// SIMATIC S7-200 project (STEP 7-Micro/WIN), CPU 224 AM REL 21.02

SYMBOL_TABLE USER1
T2SK1_TG         C1
T2SK2_TG         C2
T2SK3_TG         C3
T2SK4_TG         C4
T2SK5_TG         C5
T2SK6_TG         C6
T2SK7_TG         C7
T2SK8_TG         C8
T2SK9_TG         C9
T3SK1_TG         C10
T3SK2_TG         C11
T3SK3_TG         C12
T3SK4_TG         C13
T3SK5_TG         C14
T3SK6_TG         C15
T3SK7_TG         C16
T3SK8_TG         C17
T3SK9_TG         C18
T4SK1_TG         C19
T4SK2_TG         C20
T4SK3_TG         C21
T4SK4_TG         C22
T4SK5_TG         C23
T4SK6_TG         C24
T4SK7_TG         C25
T4SK8_TG         C26
T4SK9_TG         C27
T5SK1_TG         C28
T5SK2_TG         C29
T5SK3_TG         C30
T5SK4_TG         C31
T5SK5_TG         C32
T5SK6_TG         C33
T5SK7_TG         C34
T5SK8_TG         C35
T5SK9_TG         C36
T6SK1_TG         C37
T6SK2_TG         C38
T6SK3_TG         C39
T6SK4_TG         C40
T6SK5_TG         C41
T6SK6_TG         C42
T6SK7_TG         C43
T6SK8_TG         C44
T6SK9_TG         C45
T7SK1_TG         C46
T7SK2_TG         C47
T7SK3_TG         C48
T7SK4_TG         C49
T7SK5_TG         C50
T7SK6_TG         C51
T7SK7_TG         C52
T7SK8_TG         C53
T7SK9_TG         C54
CNSK1_TG         C55
CNSK2_TG         C56
CNSK3_TG         C57
CNSK4_TG         C58
CNSK5_TG         C59
CNSK6_TG         C60
CNSK7_TG         C61
CNSK8_TG         C62
CNSK9_TG         C63
GIO              MW0
NGAY             MW2
PHUT             MW4
THANG            MW6
THU              MW8
GIAY             MW10
AT1              Q0.0
AT2              Q0.1
AT3              Q0.2
AT4              Q0.3
AT5              Q0.4
AT6              Q0.5
AT7              Q0.6
AT8              Q0.7
TEST_1           V10.0
TEST_2           V10.1
TEST_3           V10.2
TEST_4           V10.3
TEST_5           V10.4
TEST_6           V10.5
TEST_7           V10.6
TEST_8           V10.7
T2RS             V11.2
GOI_AT           V11.3
T3RS             V11.4
T4RS             V11.5
T5RS             V11.6
T6RS             V11.7
T7RS             V12.0
CNRS             V12.1
T2SK1H           VW100
T2SK1M           VW102
T2SK1LC          VW104
T2SK1_TGD        VW106
T2SK2H           VW108
T2SK2M           VW110
T2SK2LC          VW112
T2SK2_TGD        VW114
T2SK3H           VW116
T2SK3M           VW118
T2SK3LC          VW120
T2SK3_TGD        VW122
T2SK4H           VW124
T2SK4M           VW126
T2SK4LC          VW128
T2SK4_TGD        VW130
T2SK5H           VW132
T2SK5M           VW134
T2SK5LC          VW136
T2SK5_TGD        VW138
T2SK6H           VW140
T2SK6M           VW142
T2SK6LC          VW144
T2SK6_TGD        VW146
T2SK7H           VW148
T2SK7M           VW150
T2SK7LC          VW152
T2SK7_TGD        VW154
T2SK8H           VW156
T2SK8M           VW158
T2SK8LC          VW160
T2SK8_TGD        VW162
T2SK9H           VW164
T2SK9M           VW166
T2SK9LC          VW168
T2SK9_TGD        VW170
T3SK1H           VW172
T3SK1M           VW174
T3SK1LC          VW176
T3SK1_TGD        VW178
T3SK2H           VW180
T3SK2M           VW182
T3SK2LC          VW184
T3SK2_TGD        VW186
T3SK3H           VW188
T3SK3M           VW190
T3SK3LC          VW192
T3SK3_TGD        VW194
T3SK4H           VW196
T3SK4M           VW198
T3SK4LC          VW200
T3SK4_TGD        VW202
T3SK5H           VW204
T3SK5M           VW206
T3SK5LC          VW208
T3SK5_TGD        VW210
T3SK6H           VW212
T3SK6M           VW214
T3SK6LC          VW216
T3SK6_TGD        VW218
T3SK7H           VW220
T3SK7M           VW222
T3SK7LC          VW224
T3SK7_TGD        VW226
T3SK8H           VW228
T3SK8M           VW230
T3SK8LC          VW232
T3SK8_TGD        VW234
T3SK9H           VW236
T3SK9M           VW238
T3SK9LC          VW240
T3SK9_TGD        VW242
T4SK1H           VW244
T4SK1M           VW246
T4SK1LC          VW248
T4SK1_TGD        VW250
T4SK2H           VW252
T4SK2M           VW254
T4SK2LC          VW256
T4SK2_TGD        VW258
T4SK3H           VW260
T4SK3M           VW262
T4SK3LC          VW264
T4SK3_TGD        VW266
T4SK4H           VW268
T4SK4M           VW270
T4SK4LC          VW272
T4SK4_TGD        VW274
T4SK5H           VW276
T4SK5M           VW278
T4SK5LC          VW280
T4SK5_TGD        VW282
T4SK6H           VW284
T4SK6M           VW286
T4SK6LC          VW288
T4SK6_TGD        VW290
T4SK7H           VW292
T4SK7M           VW294
T4SK7LC          VW296
T4SK7_TGD        VW298
T4SK8H           VW300
T4SK8M           VW302
T4SK8LC          VW304
T4SK8_TGD        VW306
T4SK9H           VW308
T4SK9M           VW310
T4SK9LC          VW312
T4SK9_TGD        VW314
T5SK1H           VW316
T5SK1M           VW318
T5SK1LC          VW320
T5SK1_TGD        VW322
T5SK2H           VW324
T5SK2M           VW326
T5SK2LC          VW328
T5SK2_TGD        VW330
T5SK3H           VW332
T5SK3M           VW334
T5SK3LC          VW336
T5SK3_TGD        VW338
T5SK4H           VW340
T5SK4M           VW342
T5SK4LC          VW346
T5SK4_TGD        VW348
T5SK5H           VW350
T5SK5M           VW352
T5SK5LC          VW354
T5SK5_TGD        VW356
T5SK6H           VW358
T5SK6M           VW360
T5SK6LC          VW362
T5SK6_TGD        VW364
T5SK7H           VW368
T5SK7M           VW370
T5SK7LC          VW372
T5SK7_TGD        VW374
T5SK8H           VW376
T5SK8M           VW378
T5SK8LC          VW380
T5SK8_TGD        VW382
T5SK9H           VW384
T5SK9M           VW386
T5SK9LC          VW388
T5SK9_TGD        VW390
T6SK1H           VW392
T6SK1M           VW394
T6SK1LC          VW396
T6SK1_TGD        VW398
T6SK2H           VW400
T6SK2M           VW402
T6SK2LC          VW404
T6SK2_TGD        VW406
T6SK3H           VW408
T6SK3M           VW410
T6SK3LC          VW412
T6SK3_TGD        VW414
T6SK4H           VW416
T6SK4M           VW418
T6SK4LC          VW420
T6SK4_TGD        VW422
T6SK5H           VW424
T6SK5M           VW426
T6SK5LC          VW428
T6SK5_TGD        VW430
T6SK6H           VW432
T6SK6M           VW434
T6SK6LC          VW436
T6SK6_TGD        VW438
T6SK7H           VW440
T6SK7M           VW442
T6SK7LC          VW444
T6SK7_TGD        VW446
T6SK8H           VW448
T6SK8M           VW450
T6SK8LC          VW452
T6SK8_TGD        VW454
T6SK9H           VW456
T6SK9M           VW458
T6SK9LC          VW460
T6SK9_TGD        VW462
T7SK1H           VW468
T7SK1M           VW470
T7SK1LC          VW472
T7SK1_TGD        VW474
T7SK2H           VW476
T7SK2M           VW478
T7SK2LC          VW480
T7SK2_TGD        VW482
T7SK3H           VW484
T7SK3M           VW486
T7SK3LC          VW488
T7SK3_TGD        VW490
T7SK4H           VW492
T7SK4M           VW494
T7SK4LC          VW496
T7SK4_TGD        VW498
T7SK5H           VW500
T7SK5M           VW502
T7SK5LC          VW504
T7SK5_TGD        VW506
T7SK6H           VW508
T7SK6M           VW510
T7SK6LC          VW512
T7SK6_TGD        VW514
T7SK7H           VW516
T7SK7M           VW518
T7SK7LC          VW520
T7SK7_TGD        VW522
T7SK8H           VW524
T7SK8M           VW526
T7SK8LC          VW528
T7SK8_TGD        VW530
T7SK9H           VW532
T7SK9M           VW534
T7SK9LC          VW536
T7SK9_TGD        VW538
CNSK1H           VW540
CNSK1M           VW542
CNSK1LC          VW546
CNSK1_TGD        VW548
CNSK2H           VW550
CNSK2M           VW552
CNSK2LC          VW554
CNSK2_TGD        VW556
CNSK3H           VW558
CNSK3M           VW560
CNSK3LC          VW562
CNSK3_TGD        VW564
CNSK4H           VW566
CNSK4M           VW568
CNSK4LC          VW570
CNSK4_TGD        VW572
CNSK5H           VW574
CNSK5M           VW576
CNSK5LC          VW578
CNSK5_TGD        VW580
CNSK6H           VW582
CNSK6M           VW584
CNSK6LC          VW586
CNSK6_TGD        VW588
CNSK7H           VW590
CNSK7M           VW592
CNSK7LC          VW594
CNSK7_TGD        VW596
CNSK8H           VW598
CNSK8M           VW600
CNSK8LC          VW602
CNSK8_TGD        VW604
CNSK9H           VW606
CNSK9M           VW608
CNSK9LC          VW610
CNSK9_TGD        VW612
END_SYMBOL_TABLE

ORGANIZATION_BLOCK MAIN:OB1
TITLE=PROGRAM COMMENTS
BEGIN
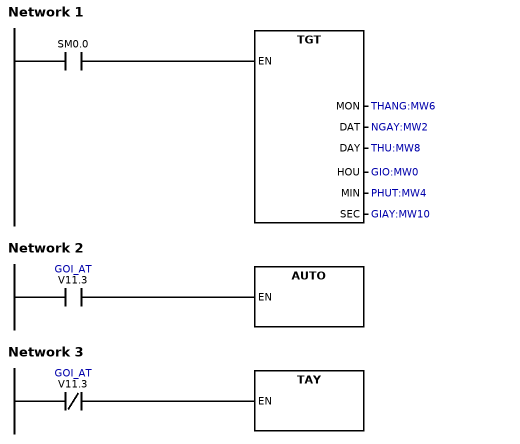
Network 1
LD     SM0.0
CALL   TGT:SBR0, THANG:MW6, NGAY:MW2, THU:MW8, GIO:MW0, PHUT:MW4, GIAY:MW10
Network 2
LD     GOI_AT:V11.3
CALL   AUTO:SBR2
Network 3
LDN    GOI_AT:V11.3
CALL   TAY:SBR1
END_ORGANIZATION_BLOCK

SUBROUTINE_BLOCK TGT:SBR0
TITLE=SUBROUTINE COMMENTS
VAR_OUTPUT
MON:INT;	// LW0 
DAT:INT;	// LW2 
DAY:INT;	// LW4 
HOU:INT;	// LW6 
MIN:INT;	// LW8 
SEC:INT;	// LW10 
END_VAR
BEGIN
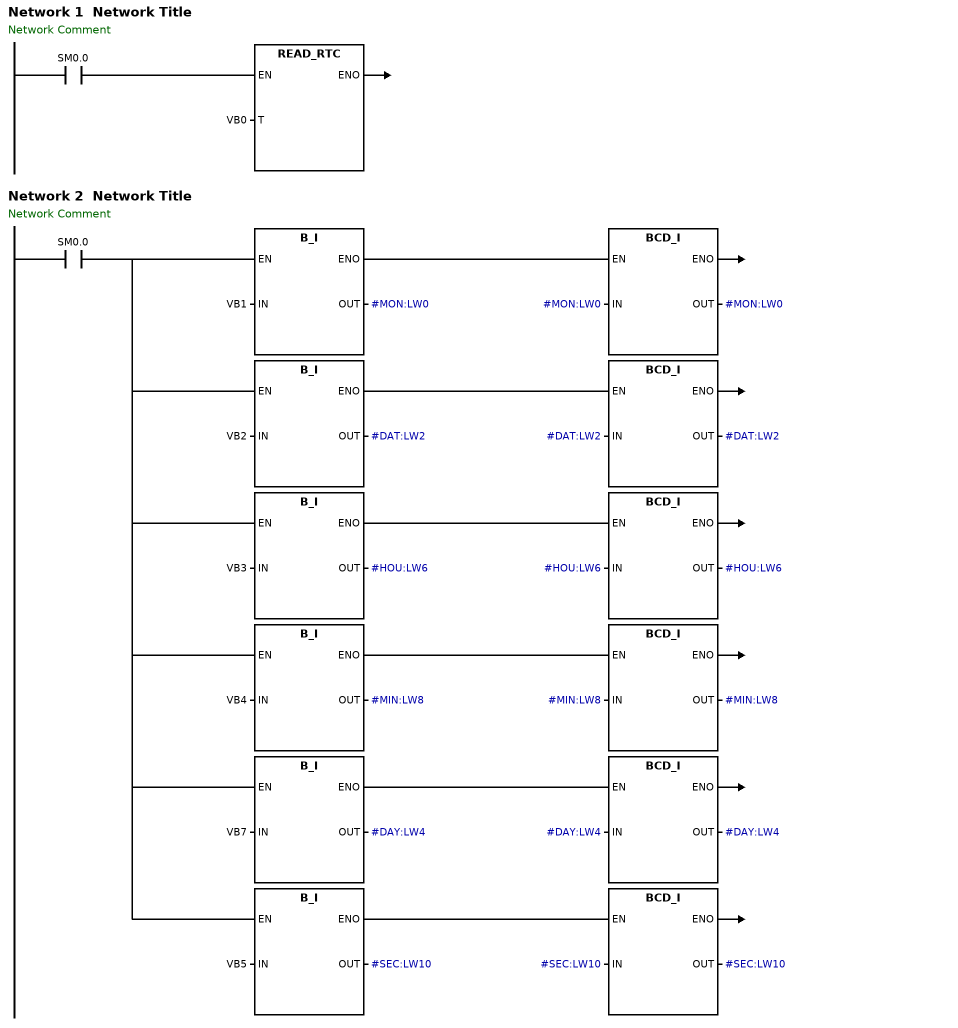
Network 1 // Network Title
// Network Comment
LD     SM0.0
TODR   VB0
Network 2 // Network Title
// Network Comment
LD     SM0.0
LPS
BTI    VB1, #MON:LW0
AENO
BCDI   #MON:LW0
LRD
BTI    VB2, #DAT:LW2
AENO
BCDI   #DAT:LW2
LRD
BTI    VB3, #HOU:LW6
AENO
BCDI   #HOU:LW6
LRD
BTI    VB4, #MIN:LW8
AENO
BCDI   #MIN:LW8
LRD
BTI    VB7, #DAY:LW4
AENO
BCDI   #DAY:LW4
LPP
BTI    VB5, #SEC:LW10
AENO
BCDI   #SEC:LW10
END_SUBROUTINE_BLOCK

SUBROUTINE_BLOCK TAY:SBR1
TITLE=SUBROUTINE COMMENTS
BEGIN
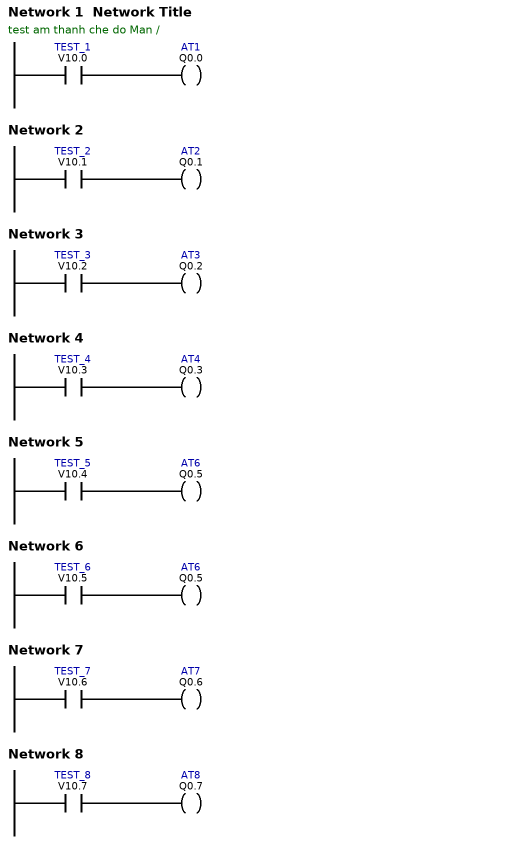
Network 1 // Network Title
// test am thanh che do Man
// 
LD     TEST_1:V10.0
=      AT1:Q0.0
Network 2
LD     TEST_2:V10.1
=      AT2:Q0.1
Network 3
LD     TEST_3:V10.2
=      AT3:Q0.2
Network 4
LD     TEST_4:V10.3
=      AT4:Q0.3
Network 5
LD     TEST_5:V10.4
=      AT6:Q0.5
Network 6
LD     TEST_6:V10.5
=      AT6:Q0.5
Network 7
LD     TEST_7:V10.6
=      AT7:Q0.6
Network 8
LD     TEST_8:V10.7
=      AT8:Q0.7
END_SUBROUTINE_BLOCK

SUBROUTINE_BLOCK AUTO:SBR2
TITLE=SUBROUTINE COMMENTS
BEGIN
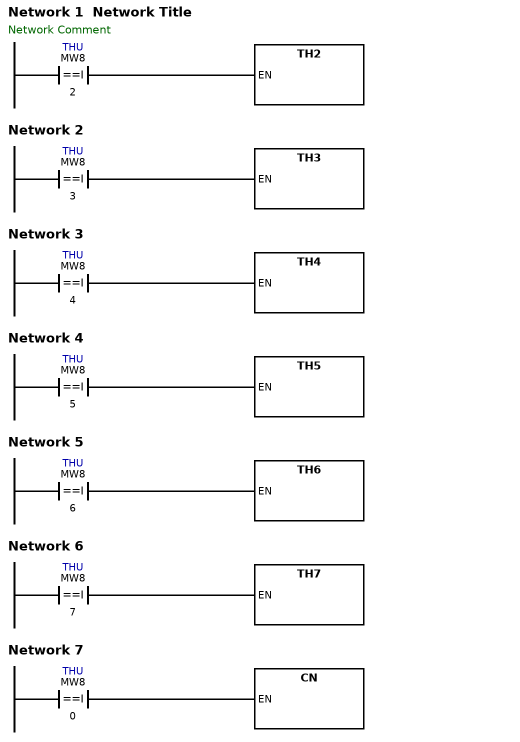
Network 1 // Network Title
// Network Comment
LDW=   THU:MW8, 2
CALL   TH2:SBR3
Network 2
LDW=   THU:MW8, 3
CALL   TH3:SBR4
Network 3
LDW=   THU:MW8, 4
CALL   TH4:SBR5
Network 4
LDW=   THU:MW8, 5
CALL   TH5:SBR6
Network 5
LDW=   THU:MW8, 6
CALL   TH6:SBR7
Network 6
LDW=   THU:MW8, 7
CALL   TH7:SBR8
Network 7
LDW=   THU:MW8, 0
CALL   CN:SBR9
END_SUBROUTINE_BLOCK

SUBROUTINE_BLOCK TH2:SBR3
TITLE=SUBROUTINE COMMENTS
VAR
TAM1:BOOL;	// L0.0 
TAM2:BOOL;	// L0.1 
TAM3:BOOL;	// L0.2 
TAM4:BOOL;	// L0.3 
TAM5:BOOL;	// L0.4 
TAM6:BOOL;	// L0.5 
TAM7:BOOL;	// L0.6 
TAM8:BOOL;	// L0.7 
TAM9:BOOL;	// L1.0 
END_VAR
BEGIN
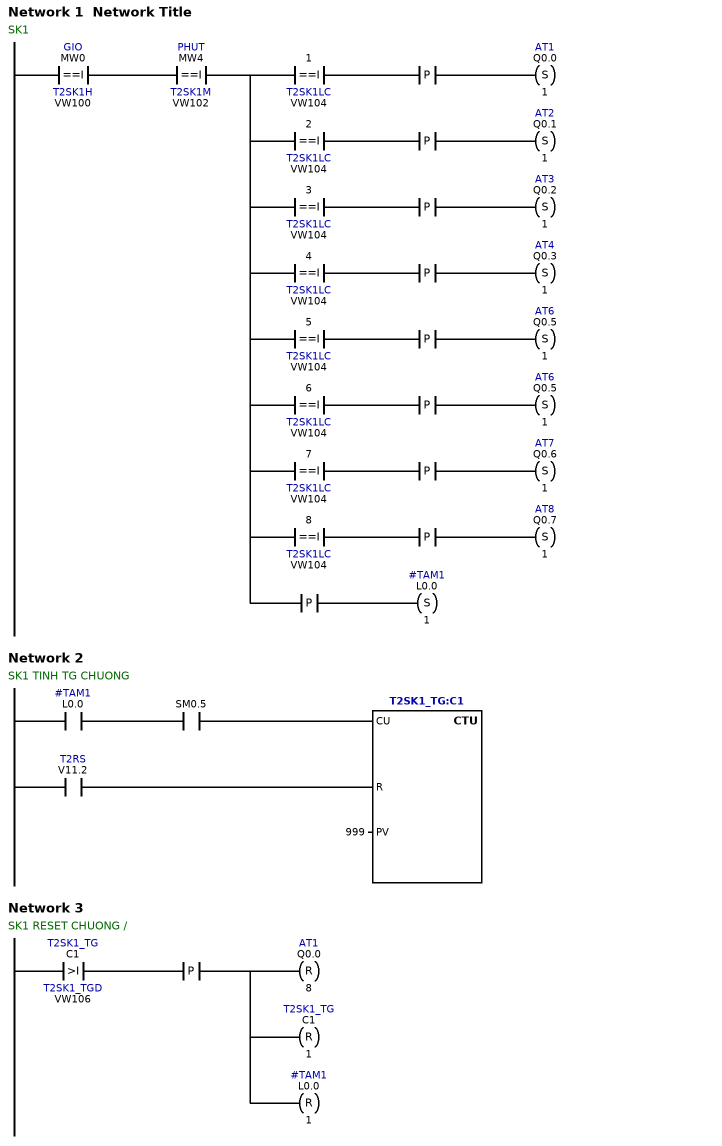
Network 1 // Network Title
// SK1	
LDW=   GIO:MW0, T2SK1H:VW100
AW=    PHUT:MW4, T2SK1M:VW102
LPS
AW=    1, T2SK1LC:VW104
EU
S      AT1:Q0.0, 1
LRD
AW=    2, T2SK1LC:VW104
EU
S      AT2:Q0.1, 1
LRD
AW=    3, T2SK1LC:VW104
EU
S      AT3:Q0.2, 1
LRD
AW=    4, T2SK1LC:VW104
EU
S      AT4:Q0.3, 1
LRD
AW=    5, T2SK1LC:VW104
EU
S      AT6:Q0.5, 1
LRD
AW=    6, T2SK1LC:VW104
EU
S      AT6:Q0.5, 1
LRD
AW=    7, T2SK1LC:VW104
EU
S      AT7:Q0.6, 1
LRD
AW=    8, T2SK1LC:VW104
EU
S      AT8:Q0.7, 1
LPP
EU
S      #TAM1:L0.0, 1
Network 2
// SK1 TINH TG CHUONG
LD     #TAM1:L0.0
A      SM0.5
LD     T2RS:V11.2
CTU    T2SK1_TG:C1, 999
Network 3
// SK1 RESET CHUONG
// 
LDW>   T2SK1_TG:C1, T2SK1_TGD:VW106
EU
R      AT1:Q0.0, 8
R      T2SK1_TG:C1, 1
R      #TAM1:L0.0, 1
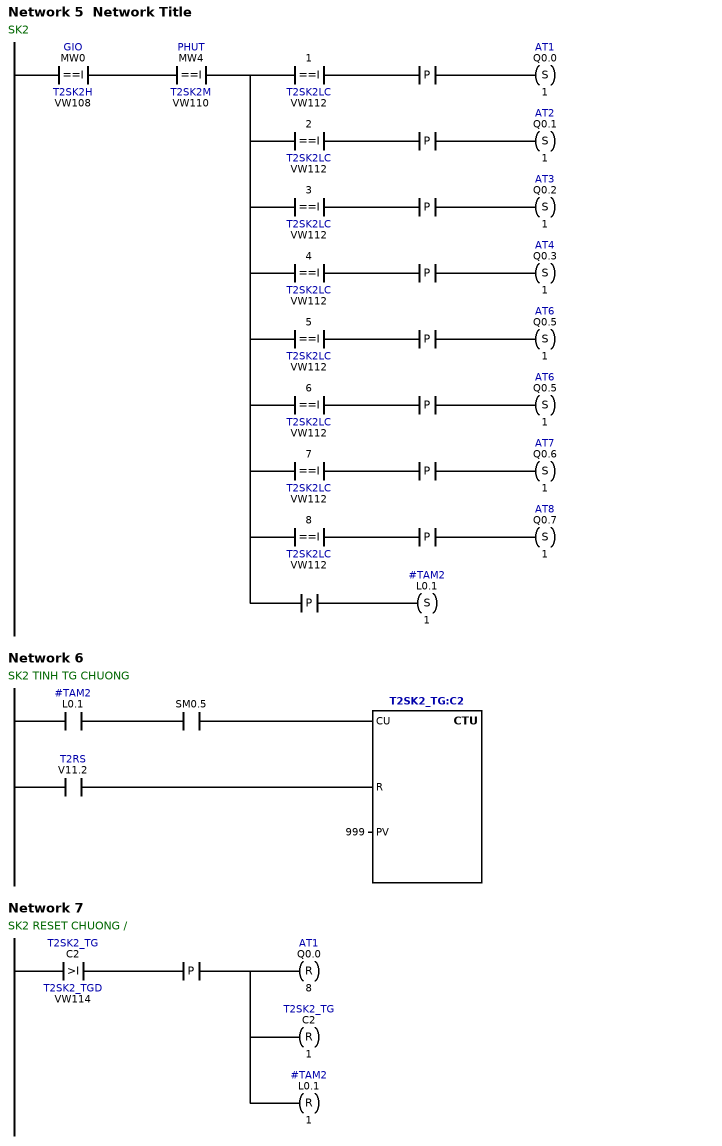
Network 5 // Network Title
// SK2
LDW=   GIO:MW0, T2SK2H:VW108
AW=    PHUT:MW4, T2SK2M:VW110
LPS
AW=    1, T2SK2LC:VW112
EU
S      AT1:Q0.0, 1
LRD
AW=    2, T2SK2LC:VW112
EU
S      AT2:Q0.1, 1
LRD
AW=    3, T2SK2LC:VW112
EU
S      AT3:Q0.2, 1
LRD
AW=    4, T2SK2LC:VW112
EU
S      AT4:Q0.3, 1
LRD
AW=    5, T2SK2LC:VW112
EU
S      AT6:Q0.5, 1
LRD
AW=    6, T2SK2LC:VW112
EU
S      AT6:Q0.5, 1
LRD
AW=    7, T2SK2LC:VW112
EU
S      AT7:Q0.6, 1
LRD
AW=    8, T2SK2LC:VW112
EU
S      AT8:Q0.7, 1
LPP
EU
S      #TAM2:L0.1, 1
Network 6
// SK2 TINH TG CHUONG
LD     #TAM2:L0.1
A      SM0.5
LD     T2RS:V11.2
CTU    T2SK2_TG:C2, 999
Network 7
// SK2 RESET CHUONG
// 
LDW>   T2SK2_TG:C2, T2SK2_TGD:VW114
EU
R      AT1:Q0.0, 8
R      T2SK2_TG:C2, 1
R      #TAM2:L0.1, 1
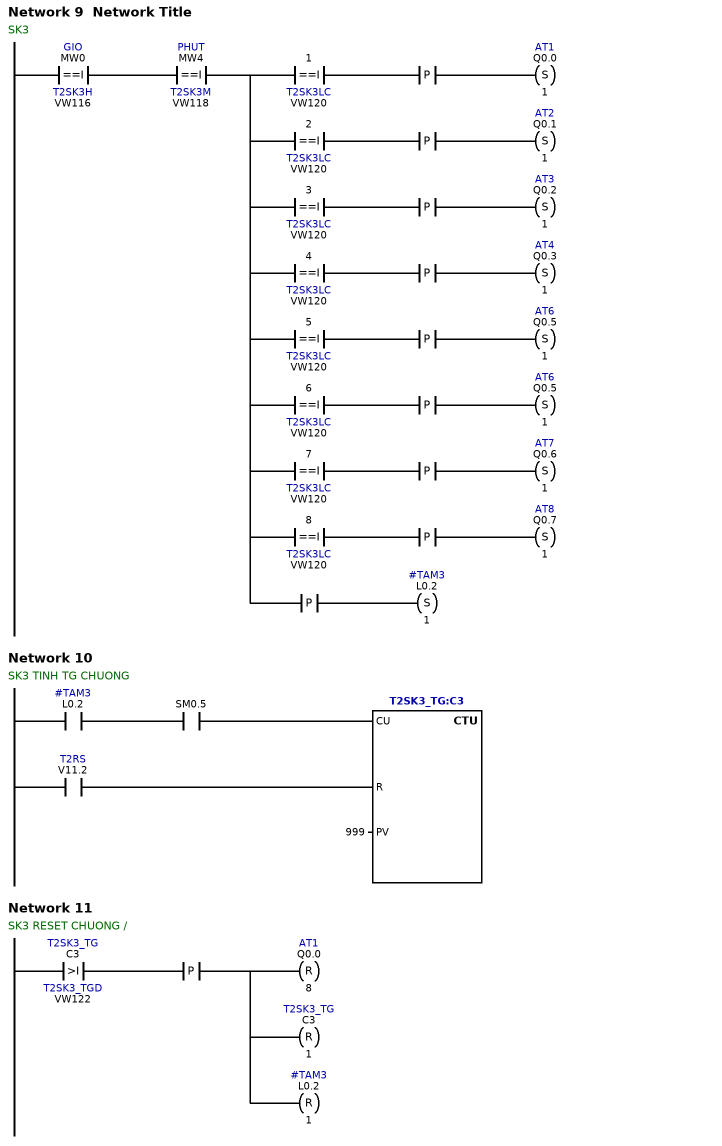
Network 9 // Network Title
// SK3	
LDW=   GIO:MW0, T2SK3H:VW116
AW=    PHUT:MW4, T2SK3M:VW118
LPS
AW=    1, T2SK3LC:VW120
EU
S      AT1:Q0.0, 1
LRD
AW=    2, T2SK3LC:VW120
EU
S      AT2:Q0.1, 1
LRD
AW=    3, T2SK3LC:VW120
EU
S      AT3:Q0.2, 1
LRD
AW=    4, T2SK3LC:VW120
EU
S      AT4:Q0.3, 1
LRD
AW=    5, T2SK3LC:VW120
EU
S      AT6:Q0.5, 1
LRD
AW=    6, T2SK3LC:VW120
EU
S      AT6:Q0.5, 1
LRD
AW=    7, T2SK3LC:VW120
EU
S      AT7:Q0.6, 1
LRD
AW=    8, T2SK3LC:VW120
EU
S      AT8:Q0.7, 1
LPP
EU
S      #TAM3:L0.2, 1
Network 10
// SK3 TINH TG CHUONG
LD     #TAM3:L0.2
A      SM0.5
LD     T2RS:V11.2
CTU    T2SK3_TG:C3, 999
Network 11
// SK3 RESET CHUONG
// 
LDW>   T2SK3_TG:C3, T2SK3_TGD:VW122
EU
R      AT1:Q0.0, 8
R      T2SK3_TG:C3, 1
R      #TAM3:L0.2, 1
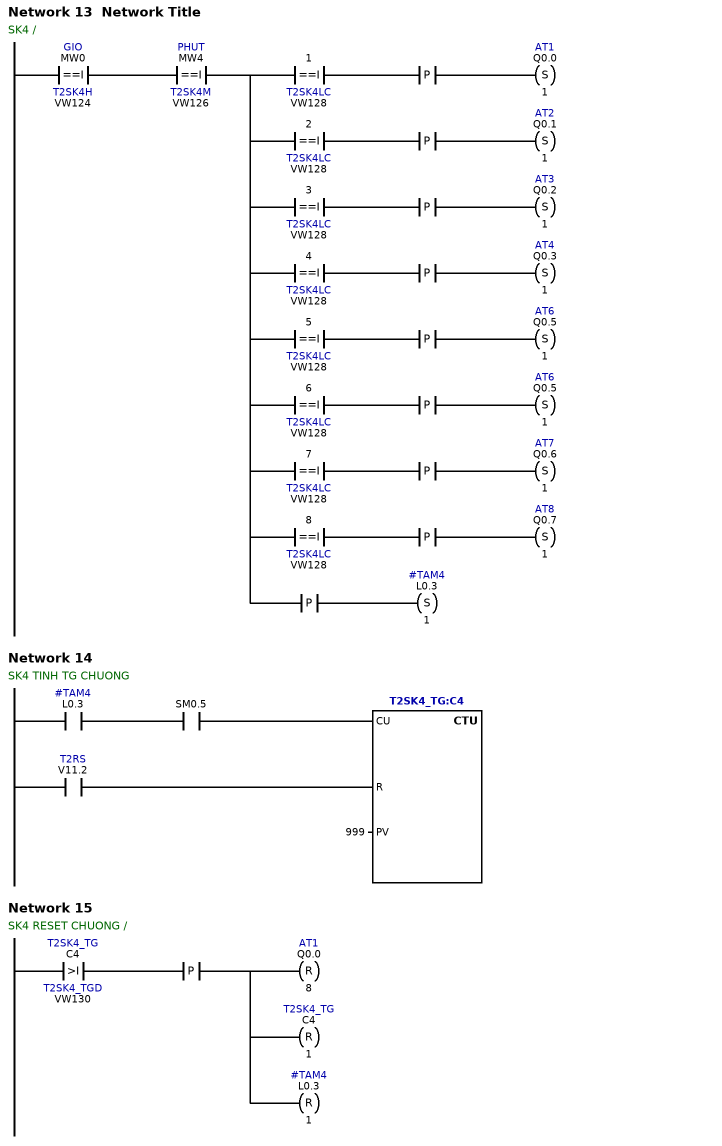
Network 13 // Network Title
// SK4
// 	
LDW=   GIO:MW0, T2SK4H:VW124
AW=    PHUT:MW4, T2SK4M:VW126
LPS
AW=    1, T2SK4LC:VW128
EU
S      AT1:Q0.0, 1
LRD
AW=    2, T2SK4LC:VW128
EU
S      AT2:Q0.1, 1
LRD
AW=    3, T2SK4LC:VW128
EU
S      AT3:Q0.2, 1
LRD
AW=    4, T2SK4LC:VW128
EU
S      AT4:Q0.3, 1
LRD
AW=    5, T2SK4LC:VW128
EU
S      AT6:Q0.5, 1
LRD
AW=    6, T2SK4LC:VW128
EU
S      AT6:Q0.5, 1
LRD
AW=    7, T2SK4LC:VW128
EU
S      AT7:Q0.6, 1
LRD
AW=    8, T2SK4LC:VW128
EU
S      AT8:Q0.7, 1
LPP
EU
S      #TAM4:L0.3, 1
Network 14
// SK4 TINH TG CHUONG
LD     #TAM4:L0.3
A      SM0.5
LD     T2RS:V11.2
CTU    T2SK4_TG:C4, 999
Network 15
// SK4 RESET CHUONG
// 
LDW>   T2SK4_TG:C4, T2SK4_TGD:VW130
EU
R      AT1:Q0.0, 8
R      T2SK4_TG:C4, 1
R      #TAM4:L0.3, 1
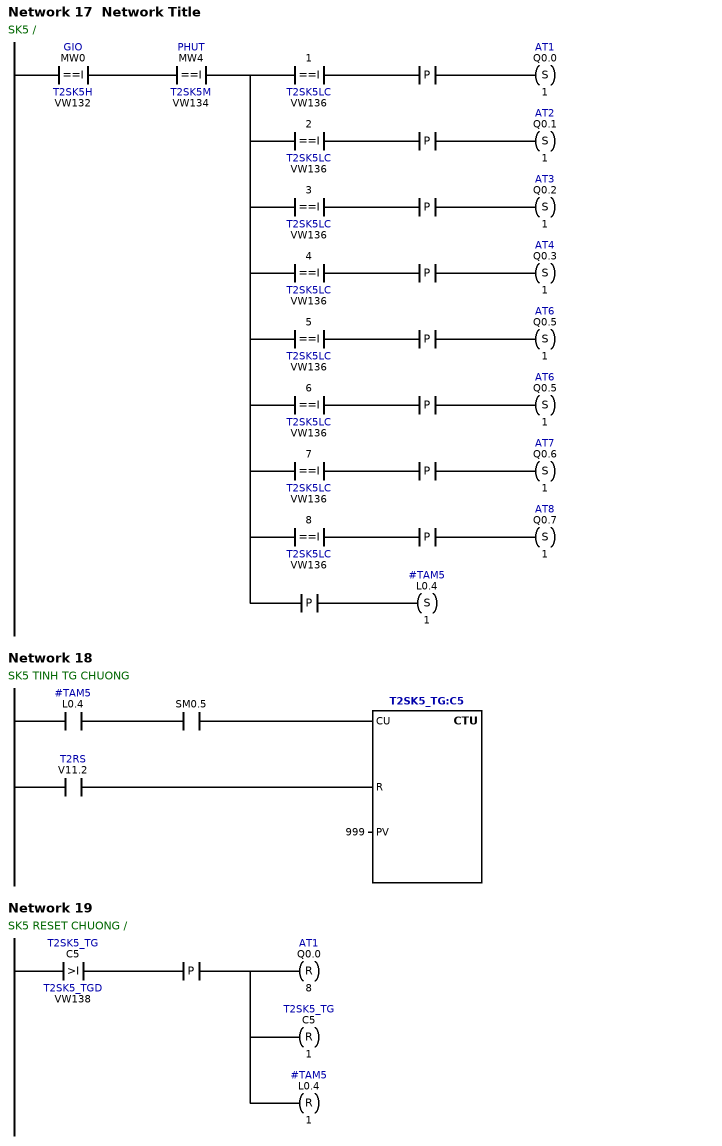
Network 17 // Network Title
// SK5
// 	
LDW=   GIO:MW0, T2SK5H:VW132
AW=    PHUT:MW4, T2SK5M:VW134
LPS
AW=    1, T2SK5LC:VW136
EU
S      AT1:Q0.0, 1
LRD
AW=    2, T2SK5LC:VW136
EU
S      AT2:Q0.1, 1
LRD
AW=    3, T2SK5LC:VW136
EU
S      AT3:Q0.2, 1
LRD
AW=    4, T2SK5LC:VW136
EU
S      AT4:Q0.3, 1
LRD
AW=    5, T2SK5LC:VW136
EU
S      AT6:Q0.5, 1
LRD
AW=    6, T2SK5LC:VW136
EU
S      AT6:Q0.5, 1
LRD
AW=    7, T2SK5LC:VW136
EU
S      AT7:Q0.6, 1
LRD
AW=    8, T2SK5LC:VW136
EU
S      AT8:Q0.7, 1
LPP
EU
S      #TAM5:L0.4, 1
Network 18
// SK5 TINH TG CHUONG
LD     #TAM5:L0.4
A      SM0.5
LD     T2RS:V11.2
CTU    T2SK5_TG:C5, 999
Network 19
// SK5 RESET CHUONG
// 
LDW>   T2SK5_TG:C5, T2SK5_TGD:VW138
EU
R      AT1:Q0.0, 8
R      T2SK5_TG:C5, 1
R      #TAM5:L0.4, 1
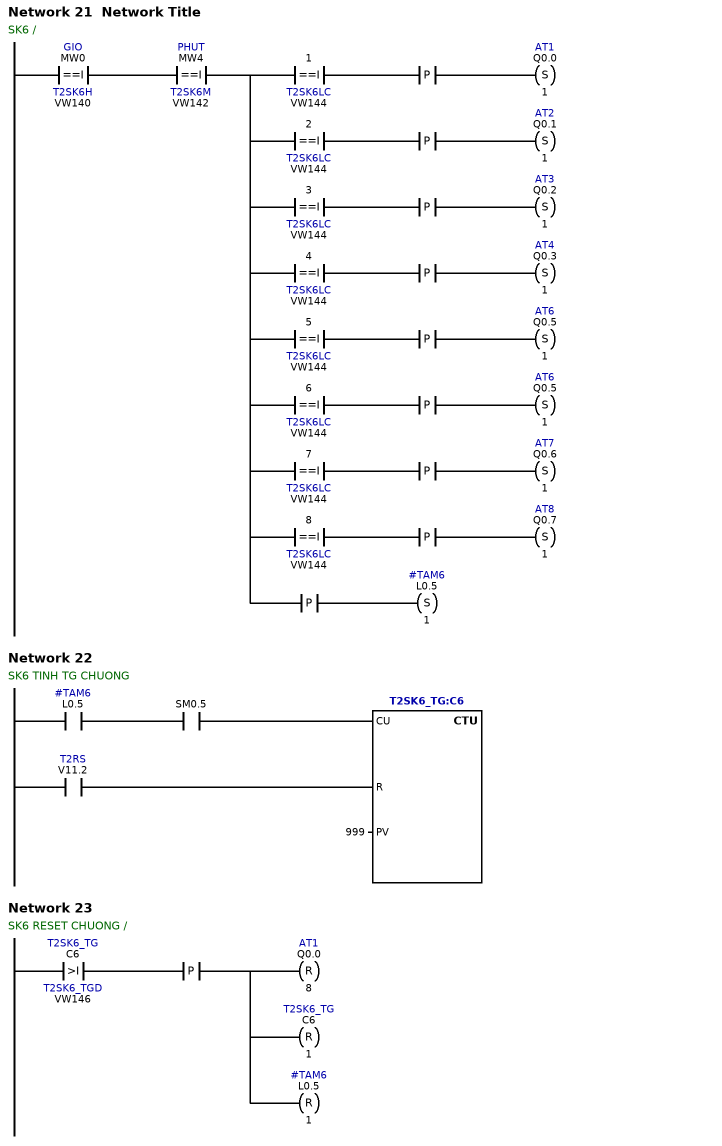
Network 21 // Network Title
// SK6
// 	
LDW=   GIO:MW0, T2SK6H:VW140
AW=    PHUT:MW4, T2SK6M:VW142
LPS
AW=    1, T2SK6LC:VW144
EU
S      AT1:Q0.0, 1
LRD
AW=    2, T2SK6LC:VW144
EU
S      AT2:Q0.1, 1
LRD
AW=    3, T2SK6LC:VW144
EU
S      AT3:Q0.2, 1
LRD
AW=    4, T2SK6LC:VW144
EU
S      AT4:Q0.3, 1
LRD
AW=    5, T2SK6LC:VW144
EU
S      AT6:Q0.5, 1
LRD
AW=    6, T2SK6LC:VW144
EU
S      AT6:Q0.5, 1
LRD
AW=    7, T2SK6LC:VW144
EU
S      AT7:Q0.6, 1
LRD
AW=    8, T2SK6LC:VW144
EU
S      AT8:Q0.7, 1
LPP
EU
S      #TAM6:L0.5, 1
Network 22
// SK6 TINH TG CHUONG
LD     #TAM6:L0.5
A      SM0.5
LD     T2RS:V11.2
CTU    T2SK6_TG:C6, 999
Network 23
// SK6 RESET CHUONG
// 
LDW>   T2SK6_TG:C6, T2SK6_TGD:VW146
EU
R      AT1:Q0.0, 8
R      T2SK6_TG:C6, 1
R      #TAM6:L0.5, 1
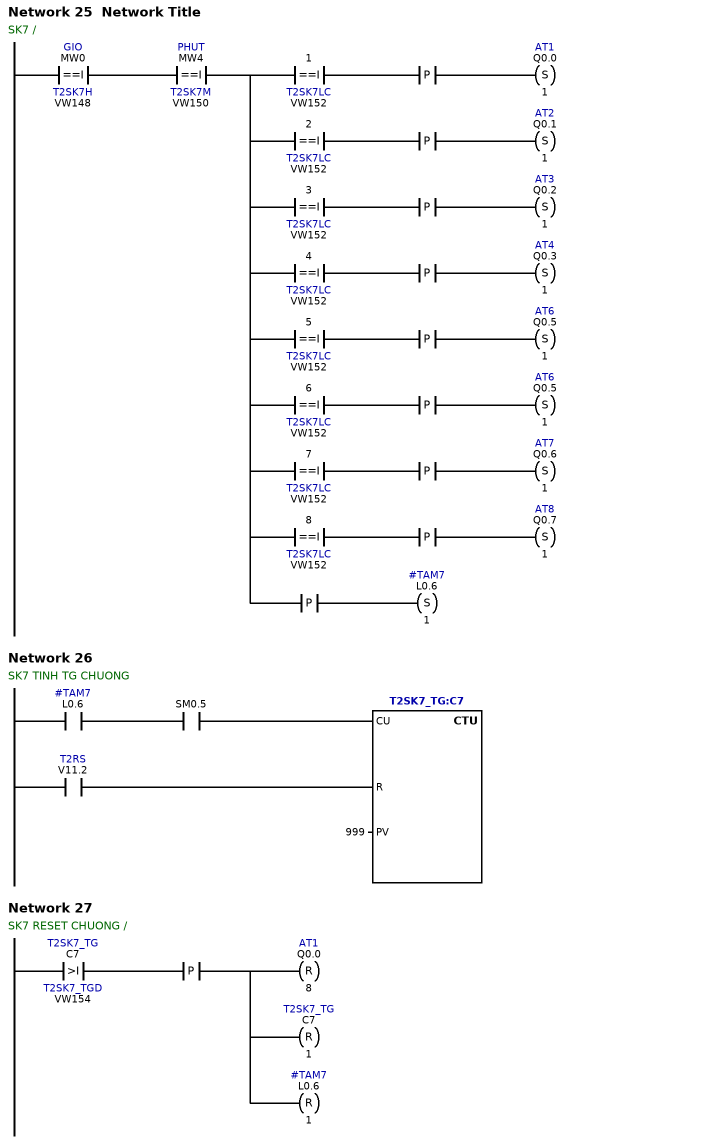
Network 25 // Network Title
// SK7
// 	
LDW=   GIO:MW0, T2SK7H:VW148
AW=    PHUT:MW4, T2SK7M:VW150
LPS
AW=    1, T2SK7LC:VW152
EU
S      AT1:Q0.0, 1
LRD
AW=    2, T2SK7LC:VW152
EU
S      AT2:Q0.1, 1
LRD
AW=    3, T2SK7LC:VW152
EU
S      AT3:Q0.2, 1
LRD
AW=    4, T2SK7LC:VW152
EU
S      AT4:Q0.3, 1
LRD
AW=    5, T2SK7LC:VW152
EU
S      AT6:Q0.5, 1
LRD
AW=    6, T2SK7LC:VW152
EU
S      AT6:Q0.5, 1
LRD
AW=    7, T2SK7LC:VW152
EU
S      AT7:Q0.6, 1
LRD
AW=    8, T2SK7LC:VW152
EU
S      AT8:Q0.7, 1
LPP
EU
S      #TAM7:L0.6, 1
Network 26
// SK7 TINH TG CHUONG
LD     #TAM7:L0.6
A      SM0.5
LD     T2RS:V11.2
CTU    T2SK7_TG:C7, 999
Network 27
// SK7 RESET CHUONG
// 
LDW>   T2SK7_TG:C7, T2SK7_TGD:VW154
EU
R      AT1:Q0.0, 8
R      T2SK7_TG:C7, 1
R      #TAM7:L0.6, 1
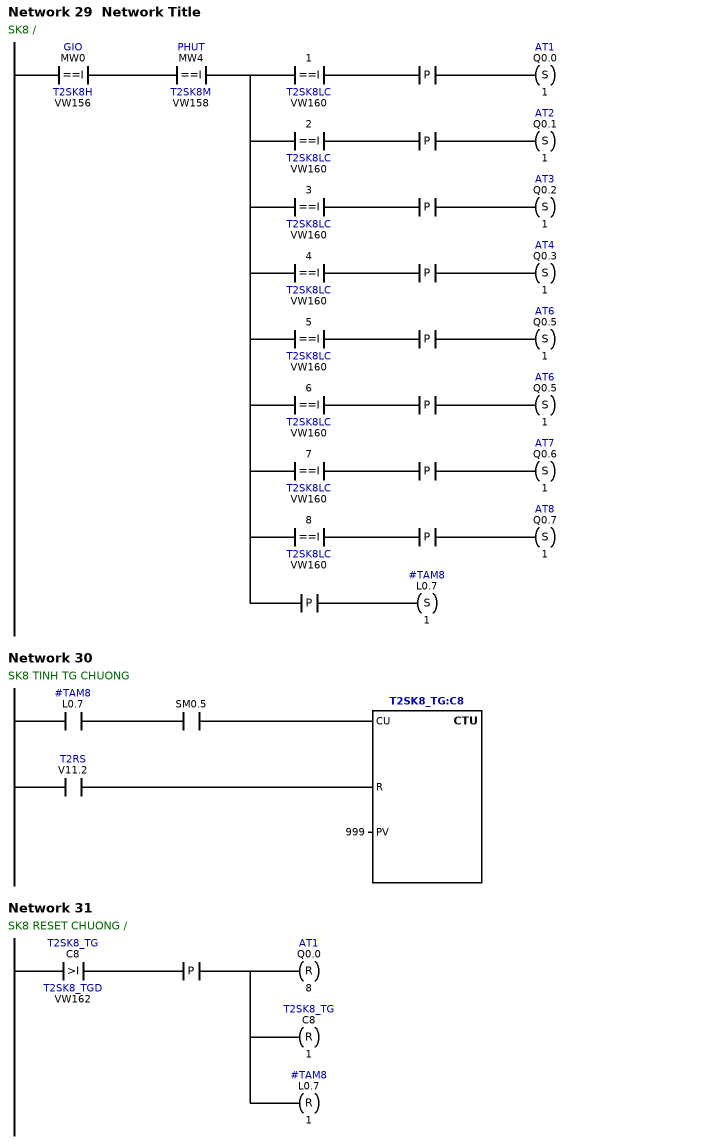
Network 29 // Network Title
// SK8
// 	
LDW=   GIO:MW0, T2SK8H:VW156
AW=    PHUT:MW4, T2SK8M:VW158
LPS
AW=    1, T2SK8LC:VW160
EU
S      AT1:Q0.0, 1
LRD
AW=    2, T2SK8LC:VW160
EU
S      AT2:Q0.1, 1
LRD
AW=    3, T2SK8LC:VW160
EU
S      AT3:Q0.2, 1
LRD
AW=    4, T2SK8LC:VW160
EU
S      AT4:Q0.3, 1
LRD
AW=    5, T2SK8LC:VW160
EU
S      AT6:Q0.5, 1
LRD
AW=    6, T2SK8LC:VW160
EU
S      AT6:Q0.5, 1
LRD
AW=    7, T2SK8LC:VW160
EU
S      AT7:Q0.6, 1
LRD
AW=    8, T2SK8LC:VW160
EU
S      AT8:Q0.7, 1
LPP
EU
S      #TAM8:L0.7, 1
Network 30
// SK8 TINH TG CHUONG
LD     #TAM8:L0.7
A      SM0.5
LD     T2RS:V11.2
CTU    T2SK8_TG:C8, 999
Network 31
// SK8 RESET CHUONG
// 
LDW>   T2SK8_TG:C8, T2SK8_TGD:VW162
EU
R      AT1:Q0.0, 8
R      T2SK8_TG:C8, 1
R      #TAM8:L0.7, 1
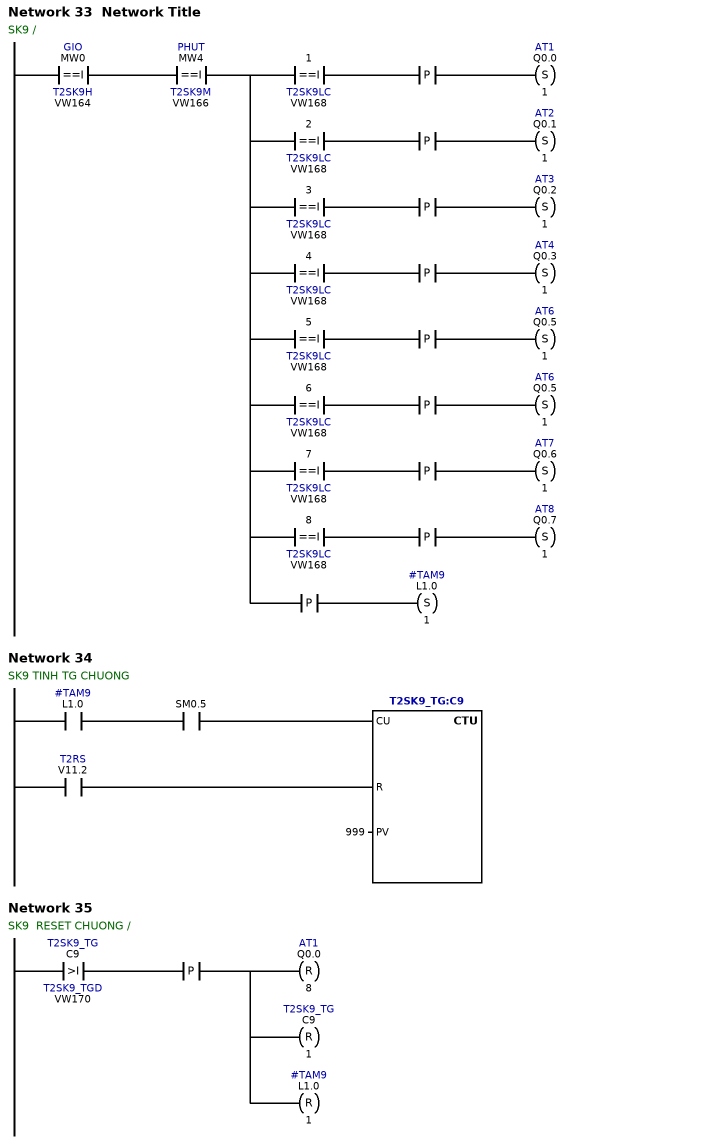
Network 33 // Network Title
// SK9
// 	
LDW=   GIO:MW0, T2SK9H:VW164
AW=    PHUT:MW4, T2SK9M:VW166
LPS
AW=    1, T2SK9LC:VW168
EU
S      AT1:Q0.0, 1
LRD
AW=    2, T2SK9LC:VW168
EU
S      AT2:Q0.1, 1
LRD
AW=    3, T2SK9LC:VW168
EU
S      AT3:Q0.2, 1
LRD
AW=    4, T2SK9LC:VW168
EU
S      AT4:Q0.3, 1
LRD
AW=    5, T2SK9LC:VW168
EU
S      AT6:Q0.5, 1
LRD
AW=    6, T2SK9LC:VW168
EU
S      AT6:Q0.5, 1
LRD
AW=    7, T2SK9LC:VW168
EU
S      AT7:Q0.6, 1
LRD
AW=    8, T2SK9LC:VW168
EU
S      AT8:Q0.7, 1
LPP
EU
S      #TAM9:L1.0, 1
Network 34
// SK9 TINH TG CHUONG
LD     #TAM9:L1.0
A      SM0.5
LD     T2RS:V11.2
CTU    T2SK9_TG:C9, 999
Network 35
// SK9  RESET CHUONG
// 
LDW>   T2SK9_TG:C9, T2SK9_TGD:VW170
EU
R      AT1:Q0.0, 8
R      T2SK9_TG:C9, 1
R      #TAM9:L1.0, 1
END_SUBROUTINE_BLOCK

SUBROUTINE_BLOCK TH3:SBR4
TITLE=SUBROUTINE COMMENTS
VAR
TAM1:BOOL;	// L0.0 
TAM2:BOOL;	// L0.1 
TAM3:BOOL;	// L0.2 
TAM4:BOOL;	// L0.3 
TAM5:BOOL;	// L0.4 
TAM6:BOOL;	// L0.5 
TAM7:BOOL;	// L0.6 
TAM8:BOOL;	// L0.7 
TAM9:BOOL;	// L1.0 
END_VAR
BEGIN
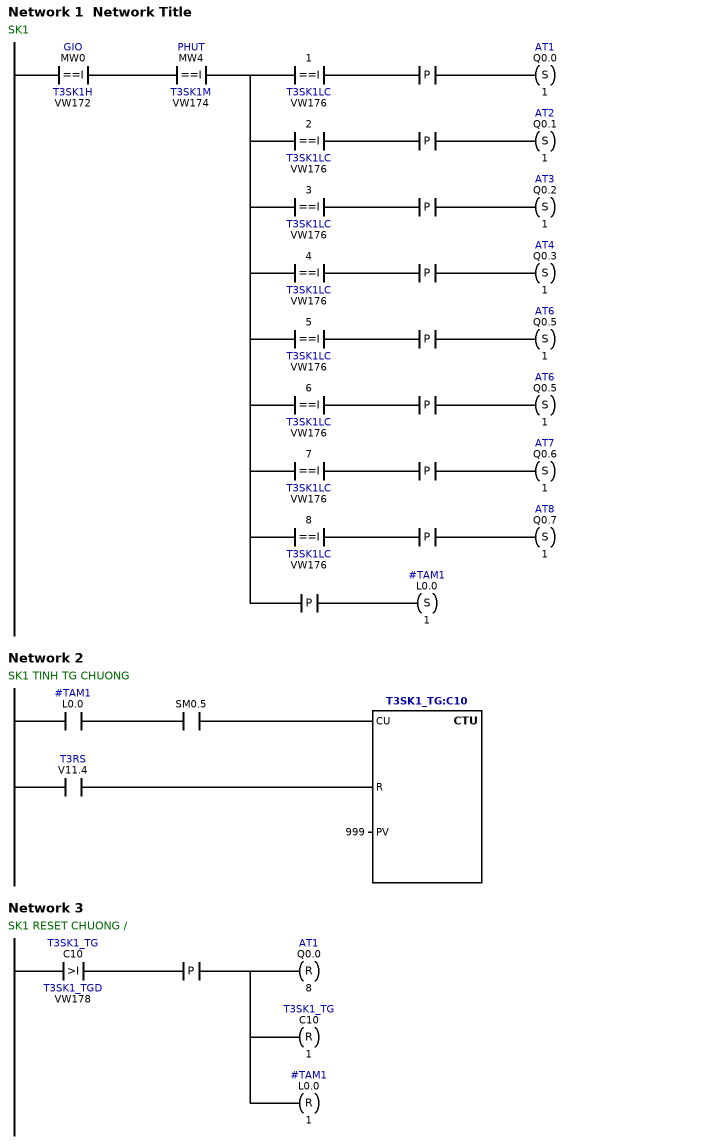
Network 1 // Network Title
// SK1	
LDW=   GIO:MW0, T3SK1H:VW172
AW=    PHUT:MW4, T3SK1M:VW174
LPS
AW=    1, T3SK1LC:VW176
EU
S      AT1:Q0.0, 1
LRD
AW=    2, T3SK1LC:VW176
EU
S      AT2:Q0.1, 1
LRD
AW=    3, T3SK1LC:VW176
EU
S      AT3:Q0.2, 1
LRD
AW=    4, T3SK1LC:VW176
EU
S      AT4:Q0.3, 1
LRD
AW=    5, T3SK1LC:VW176
EU
S      AT6:Q0.5, 1
LRD
AW=    6, T3SK1LC:VW176
EU
S      AT6:Q0.5, 1
LRD
AW=    7, T3SK1LC:VW176
EU
S      AT7:Q0.6, 1
LRD
AW=    8, T3SK1LC:VW176
EU
S      AT8:Q0.7, 1
LPP
EU
S      #TAM1:L0.0, 1
Network 2
// SK1 TINH TG CHUONG
LD     #TAM1:L0.0
A      SM0.5
LD     T3RS:V11.4
CTU    T3SK1_TG:C10, 999
Network 3
// SK1 RESET CHUONG
// 
LDW>   T3SK1_TG:C10, T3SK1_TGD:VW178
EU
R      AT1:Q0.0, 8
R      T3SK1_TG:C10, 1
R      #TAM1:L0.0, 1
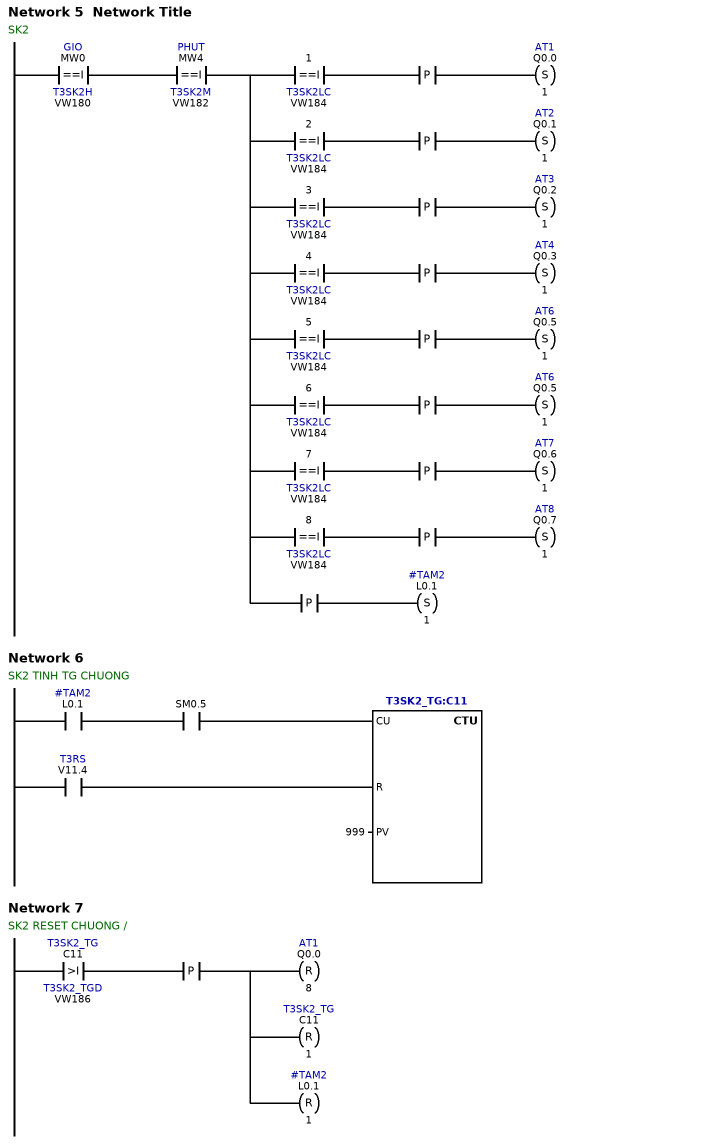
Network 5 // Network Title
// SK2
LDW=   GIO:MW0, T3SK2H:VW180
AW=    PHUT:MW4, T3SK2M:VW182
LPS
AW=    1, T3SK2LC:VW184
EU
S      AT1:Q0.0, 1
LRD
AW=    2, T3SK2LC:VW184
EU
S      AT2:Q0.1, 1
LRD
AW=    3, T3SK2LC:VW184
EU
S      AT3:Q0.2, 1
LRD
AW=    4, T3SK2LC:VW184
EU
S      AT4:Q0.3, 1
LRD
AW=    5, T3SK2LC:VW184
EU
S      AT6:Q0.5, 1
LRD
AW=    6, T3SK2LC:VW184
EU
S      AT6:Q0.5, 1
LRD
AW=    7, T3SK2LC:VW184
EU
S      AT7:Q0.6, 1
LRD
AW=    8, T3SK2LC:VW184
EU
S      AT8:Q0.7, 1
LPP
EU
S      #TAM2:L0.1, 1
Network 6
// SK2 TINH TG CHUONG
LD     #TAM2:L0.1
A      SM0.5
LD     T3RS:V11.4
CTU    T3SK2_TG:C11, 999
Network 7
// SK2 RESET CHUONG
// 
LDW>   T3SK2_TG:C11, T3SK2_TGD:VW186
EU
R      AT1:Q0.0, 8
R      T3SK2_TG:C11, 1
R      #TAM2:L0.1, 1
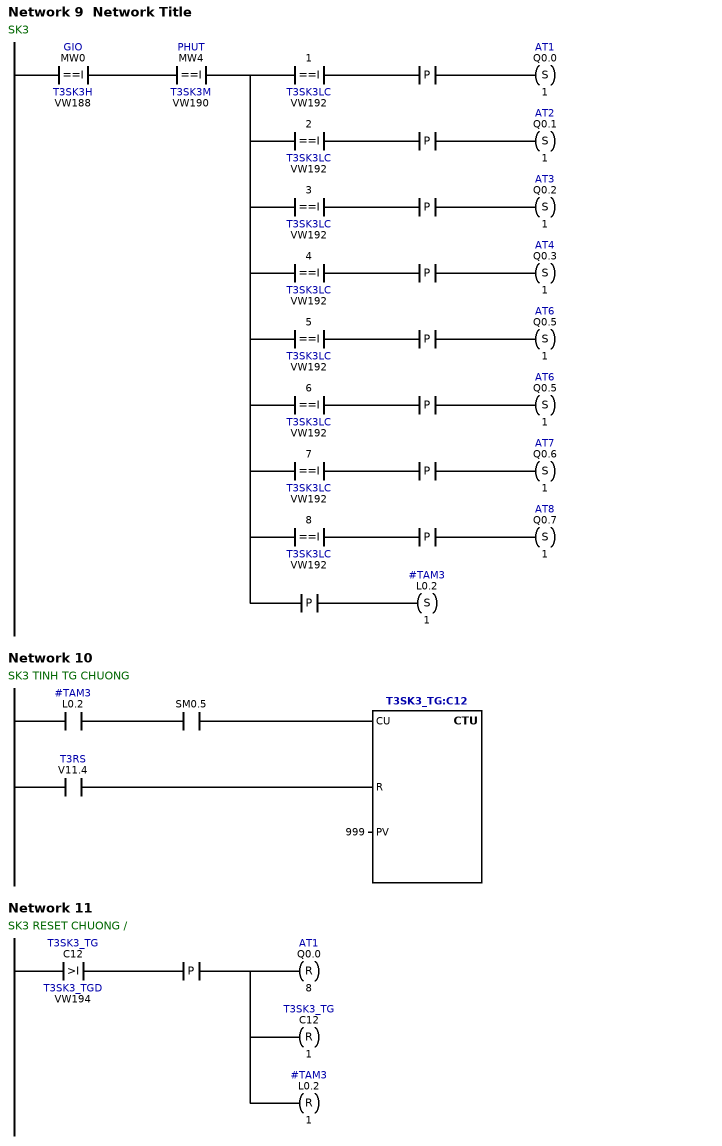
Network 9 // Network Title
// SK3	
LDW=   GIO:MW0, T3SK3H:VW188
AW=    PHUT:MW4, T3SK3M:VW190
LPS
AW=    1, T3SK3LC:VW192
EU
S      AT1:Q0.0, 1
LRD
AW=    2, T3SK3LC:VW192
EU
S      AT2:Q0.1, 1
LRD
AW=    3, T3SK3LC:VW192
EU
S      AT3:Q0.2, 1
LRD
AW=    4, T3SK3LC:VW192
EU
S      AT4:Q0.3, 1
LRD
AW=    5, T3SK3LC:VW192
EU
S      AT6:Q0.5, 1
LRD
AW=    6, T3SK3LC:VW192
EU
S      AT6:Q0.5, 1
LRD
AW=    7, T3SK3LC:VW192
EU
S      AT7:Q0.6, 1
LRD
AW=    8, T3SK3LC:VW192
EU
S      AT8:Q0.7, 1
LPP
EU
S      #TAM3:L0.2, 1
Network 10
// SK3 TINH TG CHUONG
LD     #TAM3:L0.2
A      SM0.5
LD     T3RS:V11.4
CTU    T3SK3_TG:C12, 999
Network 11
// SK3 RESET CHUONG
// 
LDW>   T3SK3_TG:C12, T3SK3_TGD:VW194
EU
R      AT1:Q0.0, 8
R      T3SK3_TG:C12, 1
R      #TAM3:L0.2, 1
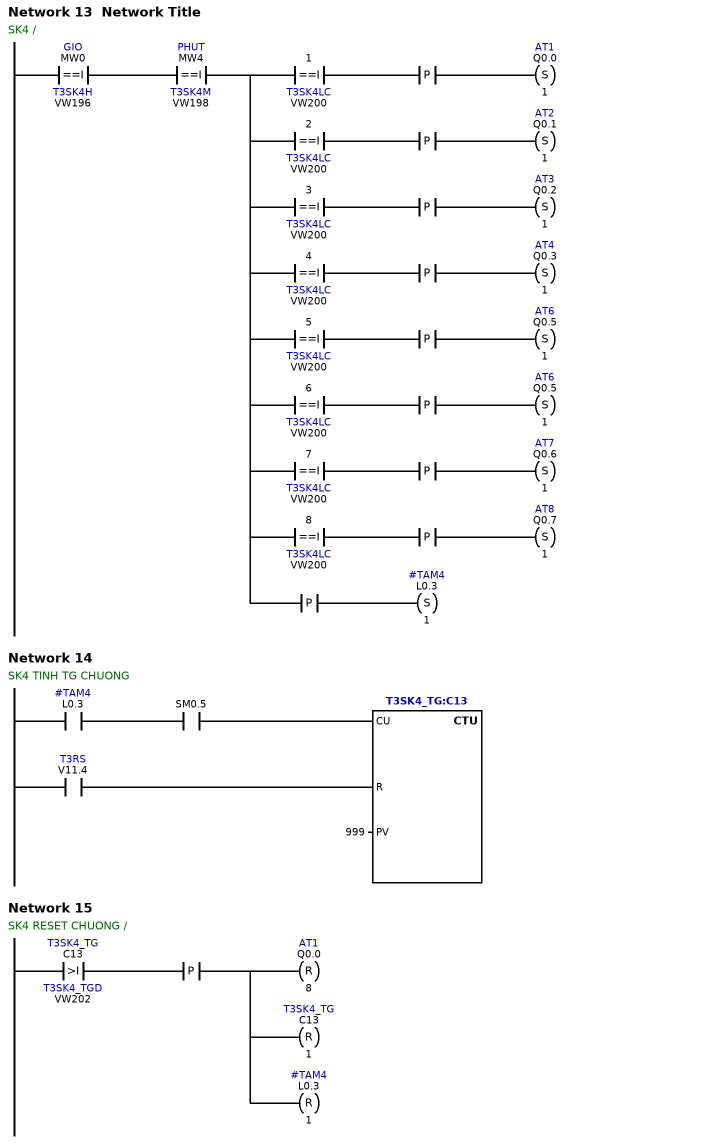
Network 13 // Network Title
// SK4
// 	
LDW=   GIO:MW0, T3SK4H:VW196
AW=    PHUT:MW4, T3SK4M:VW198
LPS
AW=    1, T3SK4LC:VW200
EU
S      AT1:Q0.0, 1
LRD
AW=    2, T3SK4LC:VW200
EU
S      AT2:Q0.1, 1
LRD
AW=    3, T3SK4LC:VW200
EU
S      AT3:Q0.2, 1
LRD
AW=    4, T3SK4LC:VW200
EU
S      AT4:Q0.3, 1
LRD
AW=    5, T3SK4LC:VW200
EU
S      AT6:Q0.5, 1
LRD
AW=    6, T3SK4LC:VW200
EU
S      AT6:Q0.5, 1
LRD
AW=    7, T3SK4LC:VW200
EU
S      AT7:Q0.6, 1
LRD
AW=    8, T3SK4LC:VW200
EU
S      AT8:Q0.7, 1
LPP
EU
S      #TAM4:L0.3, 1
Network 14
// SK4 TINH TG CHUONG
LD     #TAM4:L0.3
A      SM0.5
LD     T3RS:V11.4
CTU    T3SK4_TG:C13, 999
Network 15
// SK4 RESET CHUONG
// 
LDW>   T3SK4_TG:C13, T3SK4_TGD:VW202
EU
R      AT1:Q0.0, 8
R      T3SK4_TG:C13, 1
R      #TAM4:L0.3, 1
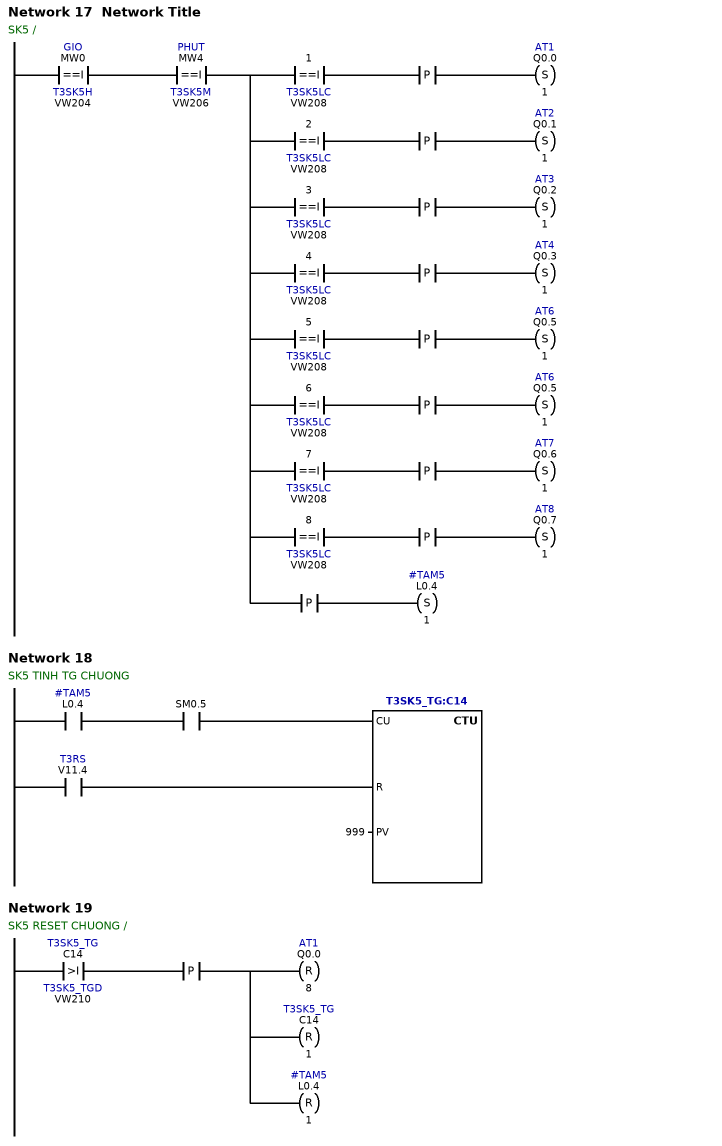
Network 17 // Network Title
// SK5
// 	
LDW=   GIO:MW0, T3SK5H:VW204
AW=    PHUT:MW4, T3SK5M:VW206
LPS
AW=    1, T3SK5LC:VW208
EU
S      AT1:Q0.0, 1
LRD
AW=    2, T3SK5LC:VW208
EU
S      AT2:Q0.1, 1
LRD
AW=    3, T3SK5LC:VW208
EU
S      AT3:Q0.2, 1
LRD
AW=    4, T3SK5LC:VW208
EU
S      AT4:Q0.3, 1
LRD
AW=    5, T3SK5LC:VW208
EU
S      AT6:Q0.5, 1
LRD
AW=    6, T3SK5LC:VW208
EU
S      AT6:Q0.5, 1
LRD
AW=    7, T3SK5LC:VW208
EU
S      AT7:Q0.6, 1
LRD
AW=    8, T3SK5LC:VW208
EU
S      AT8:Q0.7, 1
LPP
EU
S      #TAM5:L0.4, 1
Network 18
// SK5 TINH TG CHUONG
LD     #TAM5:L0.4
A      SM0.5
LD     T3RS:V11.4
CTU    T3SK5_TG:C14, 999
Network 19
// SK5 RESET CHUONG
// 
LDW>   T3SK5_TG:C14, T3SK5_TGD:VW210
EU
R      AT1:Q0.0, 8
R      T3SK5_TG:C14, 1
R      #TAM5:L0.4, 1
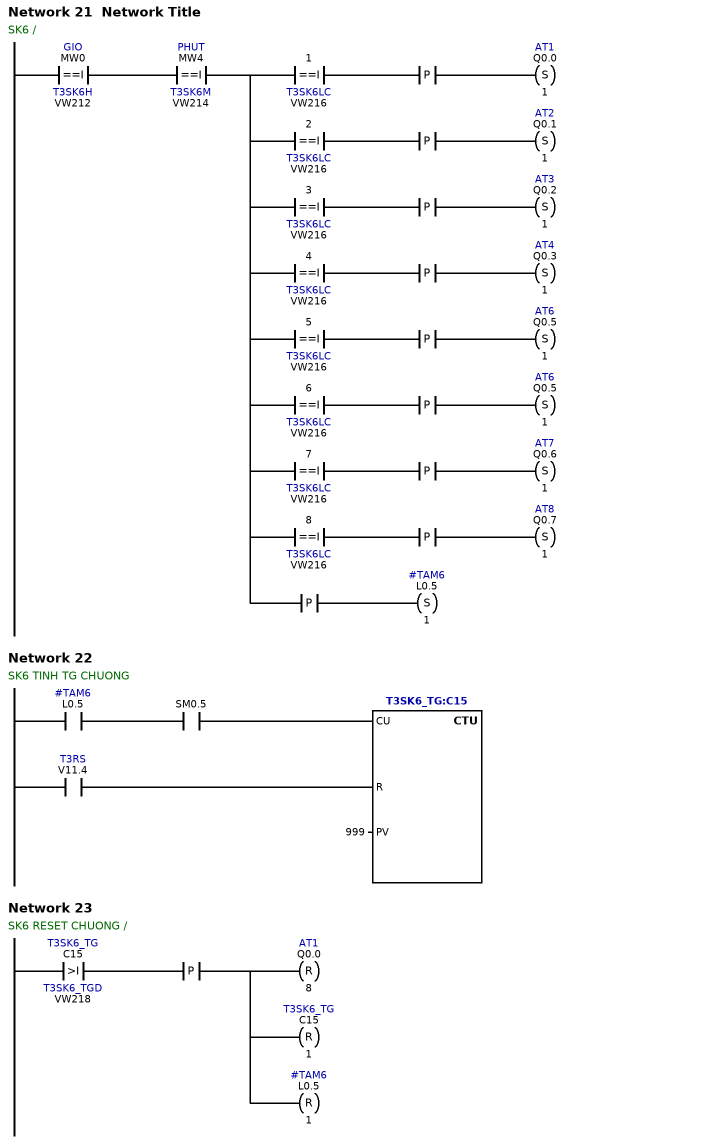
Network 21 // Network Title
// SK6
// 	
LDW=   GIO:MW0, T3SK6H:VW212
AW=    PHUT:MW4, T3SK6M:VW214
LPS
AW=    1, T3SK6LC:VW216
EU
S      AT1:Q0.0, 1
LRD
AW=    2, T3SK6LC:VW216
EU
S      AT2:Q0.1, 1
LRD
AW=    3, T3SK6LC:VW216
EU
S      AT3:Q0.2, 1
LRD
AW=    4, T3SK6LC:VW216
EU
S      AT4:Q0.3, 1
LRD
AW=    5, T3SK6LC:VW216
EU
S      AT6:Q0.5, 1
LRD
AW=    6, T3SK6LC:VW216
EU
S      AT6:Q0.5, 1
LRD
AW=    7, T3SK6LC:VW216
EU
S      AT7:Q0.6, 1
LRD
AW=    8, T3SK6LC:VW216
EU
S      AT8:Q0.7, 1
LPP
EU
S      #TAM6:L0.5, 1
Network 22
// SK6 TINH TG CHUONG
LD     #TAM6:L0.5
A      SM0.5
LD     T3RS:V11.4
CTU    T3SK6_TG:C15, 999
Network 23
// SK6 RESET CHUONG
// 
LDW>   T3SK6_TG:C15, T3SK6_TGD:VW218
EU
R      AT1:Q0.0, 8
R      T3SK6_TG:C15, 1
R      #TAM6:L0.5, 1
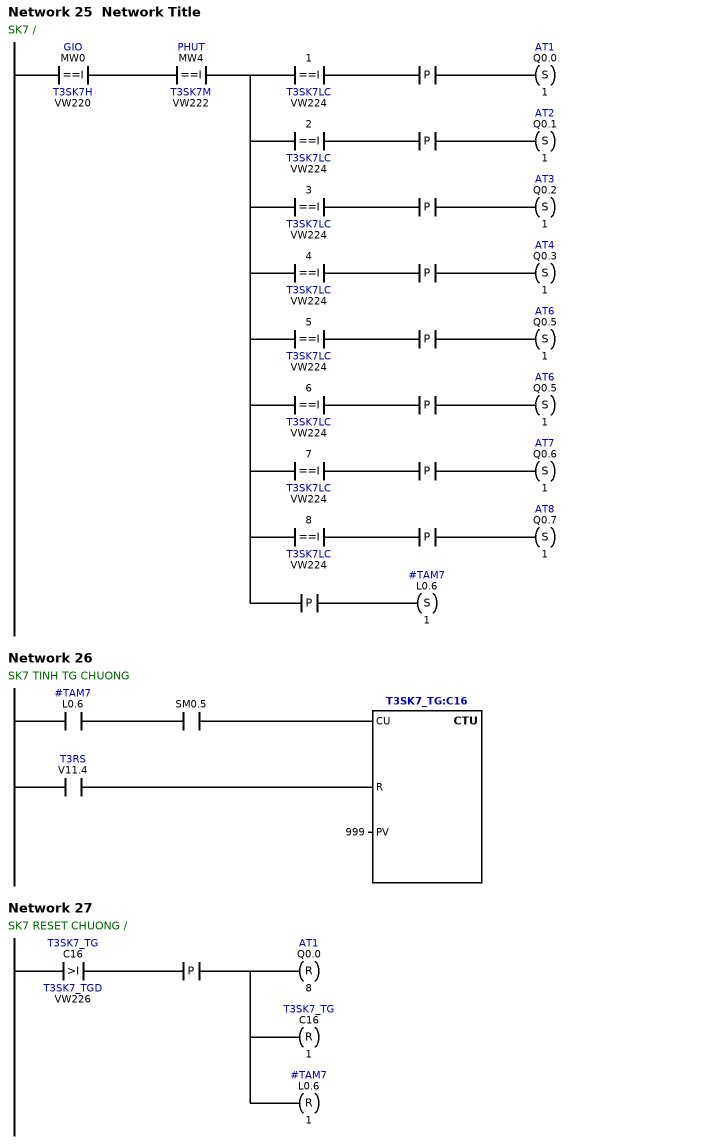
Network 25 // Network Title
// SK7
// 	
LDW=   GIO:MW0, T3SK7H:VW220
AW=    PHUT:MW4, T3SK7M:VW222
LPS
AW=    1, T3SK7LC:VW224
EU
S      AT1:Q0.0, 1
LRD
AW=    2, T3SK7LC:VW224
EU
S      AT2:Q0.1, 1
LRD
AW=    3, T3SK7LC:VW224
EU
S      AT3:Q0.2, 1
LRD
AW=    4, T3SK7LC:VW224
EU
S      AT4:Q0.3, 1
LRD
AW=    5, T3SK7LC:VW224
EU
S      AT6:Q0.5, 1
LRD
AW=    6, T3SK7LC:VW224
EU
S      AT6:Q0.5, 1
LRD
AW=    7, T3SK7LC:VW224
EU
S      AT7:Q0.6, 1
LRD
AW=    8, T3SK7LC:VW224
EU
S      AT8:Q0.7, 1
LPP
EU
S      #TAM7:L0.6, 1
Network 26
// SK7 TINH TG CHUONG
LD     #TAM7:L0.6
A      SM0.5
LD     T3RS:V11.4
CTU    T3SK7_TG:C16, 999
Network 27
// SK7 RESET CHUONG
// 
LDW>   T3SK7_TG:C16, T3SK7_TGD:VW226
EU
R      AT1:Q0.0, 8
R      T3SK7_TG:C16, 1
R      #TAM7:L0.6, 1
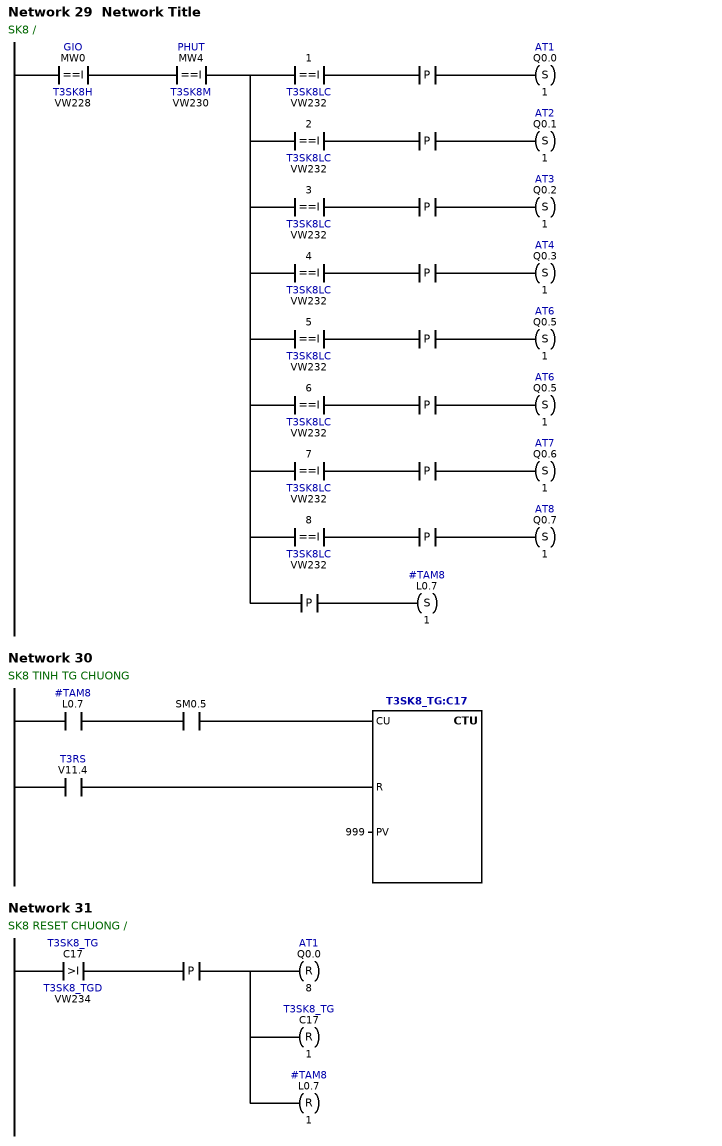
Network 29 // Network Title
// SK8
// 	
LDW=   GIO:MW0, T3SK8H:VW228
AW=    PHUT:MW4, T3SK8M:VW230
LPS
AW=    1, T3SK8LC:VW232
EU
S      AT1:Q0.0, 1
LRD
AW=    2, T3SK8LC:VW232
EU
S      AT2:Q0.1, 1
LRD
AW=    3, T3SK8LC:VW232
EU
S      AT3:Q0.2, 1
LRD
AW=    4, T3SK8LC:VW232
EU
S      AT4:Q0.3, 1
LRD
AW=    5, T3SK8LC:VW232
EU
S      AT6:Q0.5, 1
LRD
AW=    6, T3SK8LC:VW232
EU
S      AT6:Q0.5, 1
LRD
AW=    7, T3SK8LC:VW232
EU
S      AT7:Q0.6, 1
LRD
AW=    8, T3SK8LC:VW232
EU
S      AT8:Q0.7, 1
LPP
EU
S      #TAM8:L0.7, 1
Network 30
// SK8 TINH TG CHUONG
LD     #TAM8:L0.7
A      SM0.5
LD     T3RS:V11.4
CTU    T3SK8_TG:C17, 999
Network 31
// SK8 RESET CHUONG
// 
LDW>   T3SK8_TG:C17, T3SK8_TGD:VW234
EU
R      AT1:Q0.0, 8
R      T3SK8_TG:C17, 1
R      #TAM8:L0.7, 1
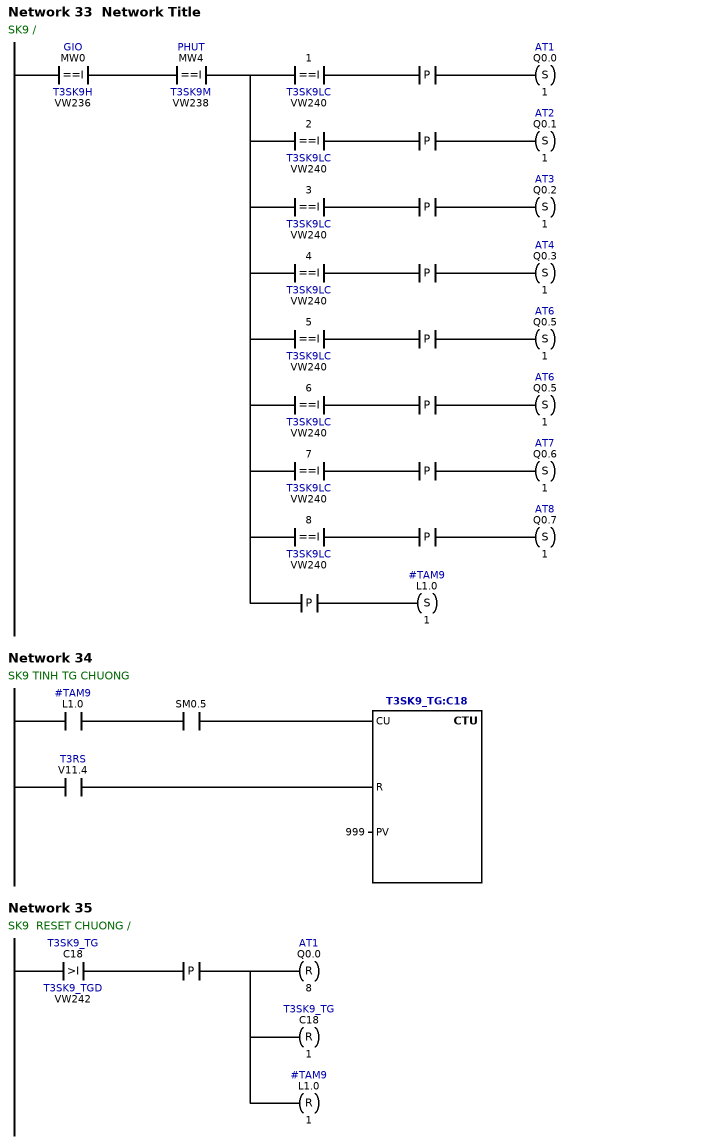
Network 33 // Network Title
// SK9
// 	
LDW=   GIO:MW0, T3SK9H:VW236
AW=    PHUT:MW4, T3SK9M:VW238
LPS
AW=    1, T3SK9LC:VW240
EU
S      AT1:Q0.0, 1
LRD
AW=    2, T3SK9LC:VW240
EU
S      AT2:Q0.1, 1
LRD
AW=    3, T3SK9LC:VW240
EU
S      AT3:Q0.2, 1
LRD
AW=    4, T3SK9LC:VW240
EU
S      AT4:Q0.3, 1
LRD
AW=    5, T3SK9LC:VW240
EU
S      AT6:Q0.5, 1
LRD
AW=    6, T3SK9LC:VW240
EU
S      AT6:Q0.5, 1
LRD
AW=    7, T3SK9LC:VW240
EU
S      AT7:Q0.6, 1
LRD
AW=    8, T3SK9LC:VW240
EU
S      AT8:Q0.7, 1
LPP
EU
S      #TAM9:L1.0, 1
Network 34
// SK9 TINH TG CHUONG
LD     #TAM9:L1.0
A      SM0.5
LD     T3RS:V11.4
CTU    T3SK9_TG:C18, 999
Network 35
// SK9  RESET CHUONG
// 
LDW>   T3SK9_TG:C18, T3SK9_TGD:VW242
EU
R      AT1:Q0.0, 8
R      T3SK9_TG:C18, 1
R      #TAM9:L1.0, 1
Network 43 // Network Title
// Network Comment
END_SUBROUTINE_BLOCK

SUBROUTINE_BLOCK TH4:SBR5
TITLE=SUBROUTINE COMMENTS
VAR
TAM1:BOOL;	// L0.0 
TAM2:BOOL;	// L0.1 
TAM3:BOOL;	// L0.2 
TAM4:BOOL;	// L0.3 
TAM5:BOOL;	// L0.4 
TAM6:BOOL;	// L0.5 
TAM7:BOOL;	// L0.6 
TAM8:BOOL;	// L0.7 
TAM9:BOOL;	// L1.0 
END_VAR
BEGIN
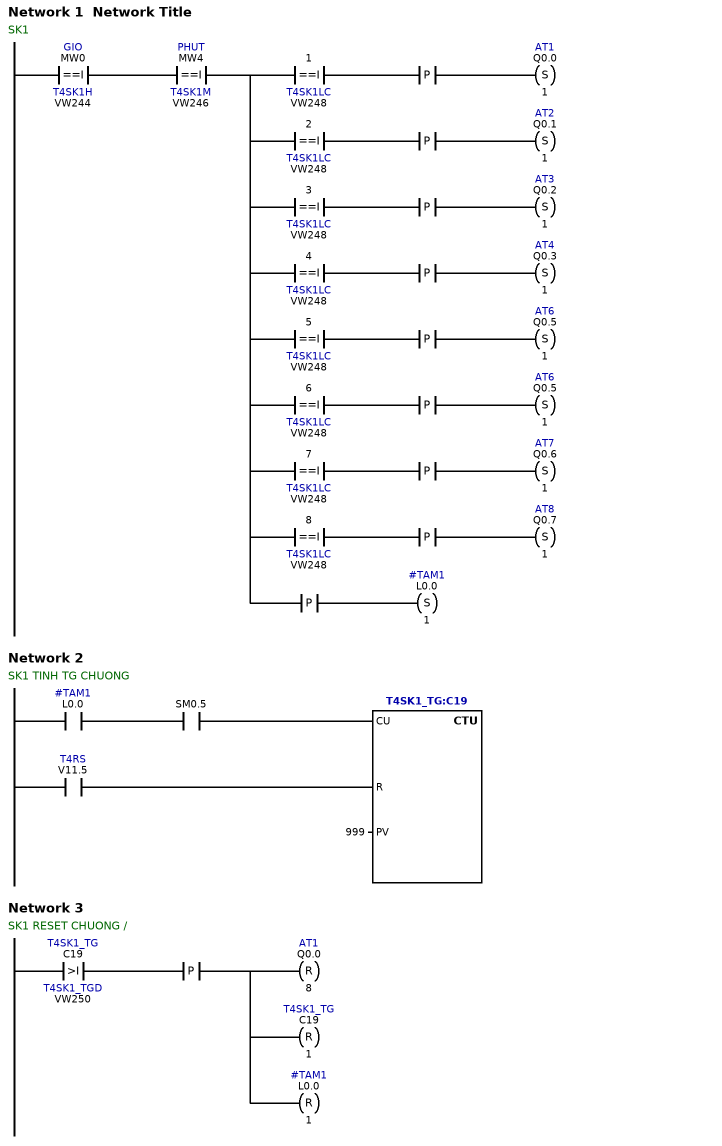
Network 1 // Network Title
// SK1	
LDW=   GIO:MW0, T4SK1H:VW244
AW=    PHUT:MW4, T4SK1M:VW246
LPS
AW=    1, T4SK1LC:VW248
EU
S      AT1:Q0.0, 1
LRD
AW=    2, T4SK1LC:VW248
EU
S      AT2:Q0.1, 1
LRD
AW=    3, T4SK1LC:VW248
EU
S      AT3:Q0.2, 1
LRD
AW=    4, T4SK1LC:VW248
EU
S      AT4:Q0.3, 1
LRD
AW=    5, T4SK1LC:VW248
EU
S      AT6:Q0.5, 1
LRD
AW=    6, T4SK1LC:VW248
EU
S      AT6:Q0.5, 1
LRD
AW=    7, T4SK1LC:VW248
EU
S      AT7:Q0.6, 1
LRD
AW=    8, T4SK1LC:VW248
EU
S      AT8:Q0.7, 1
LPP
EU
S      #TAM1:L0.0, 1
Network 2
// SK1 TINH TG CHUONG
LD     #TAM1:L0.0
A      SM0.5
LD     T4RS:V11.5
CTU    T4SK1_TG:C19, 999
Network 3
// SK1 RESET CHUONG
// 
LDW>   T4SK1_TG:C19, T4SK1_TGD:VW250
EU
R      AT1:Q0.0, 8
R      T4SK1_TG:C19, 1
R      #TAM1:L0.0, 1
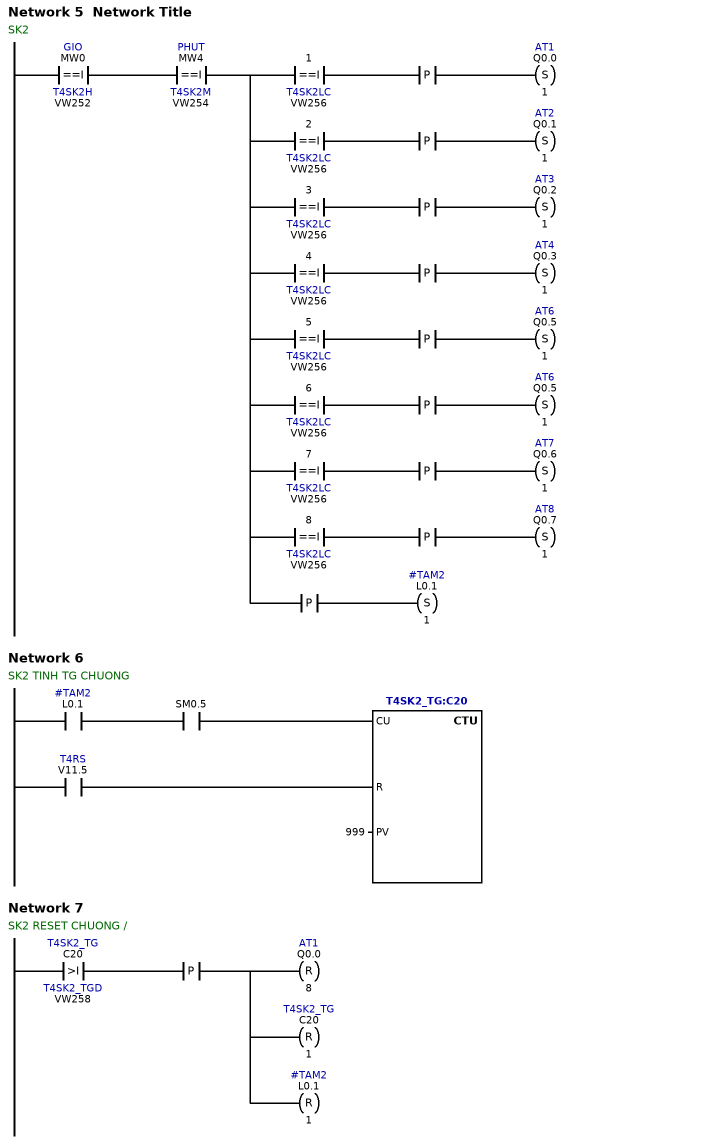
Network 5 // Network Title
// SK2
LDW=   GIO:MW0, T4SK2H:VW252
AW=    PHUT:MW4, T4SK2M:VW254
LPS
AW=    1, T4SK2LC:VW256
EU
S      AT1:Q0.0, 1
LRD
AW=    2, T4SK2LC:VW256
EU
S      AT2:Q0.1, 1
LRD
AW=    3, T4SK2LC:VW256
EU
S      AT3:Q0.2, 1
LRD
AW=    4, T4SK2LC:VW256
EU
S      AT4:Q0.3, 1
LRD
AW=    5, T4SK2LC:VW256
EU
S      AT6:Q0.5, 1
LRD
AW=    6, T4SK2LC:VW256
EU
S      AT6:Q0.5, 1
LRD
AW=    7, T4SK2LC:VW256
EU
S      AT7:Q0.6, 1
LRD
AW=    8, T4SK2LC:VW256
EU
S      AT8:Q0.7, 1
LPP
EU
S      #TAM2:L0.1, 1
Network 6
// SK2 TINH TG CHUONG
LD     #TAM2:L0.1
A      SM0.5
LD     T4RS:V11.5
CTU    T4SK2_TG:C20, 999
Network 7
// SK2 RESET CHUONG
// 
LDW>   T4SK2_TG:C20, T4SK2_TGD:VW258
EU
R      AT1:Q0.0, 8
R      T4SK2_TG:C20, 1
R      #TAM2:L0.1, 1
